// TIA Portal V20 export
TYPE "LConSMC_typeSectionalDriveOutput"
// stored: Access Published
   STRUCT
      busy : Bool := FALSE;   // TRUE : Der Funktionsbaustein wird ausgeführt / TRUE : Function block is executed
      active : Bool := FALSE;   // TRUE: Es werden Sollwerte an den Antrieb gesendet / TRUE: Setpoints are send to the drive
      ctrlBusy : Bool := FALSE;   // TRUE: Bahnzugregelung ist aktiv / TRUE: Tension control is active
      inSync : Bool;   // TRUE: Der Antrieb hat die Bahngeschwindigkeit erreicht und ist synchron / TRUE: The drive has reached the web velocity and is synchronous
      error : Bool := FALSE;   // TRUE: Es ist ein Fehler aufgetreten / TRUE: Function block has detected an error
      errorID : DWord := 16#0000_0000;   // Weiteren Informationen zu aufgetretenem Fehler (<> 16#0000_0000) / Further information on occured error (<> 16#0000_0000)
   END_STRUCT;
END_TYPE
